{attribute 'pack_mode' := '2'}
TYPE ST_CAM_CTRL :
STRUCT
  eCtrl               : E_AXIS_CTRL;    // commanded axis function
  eProgress           : E_PROGRESS;     // progress command for synced functions
END_STRUCT
END_TYPE

(* stored: Version 1.1.0.1, ProductVersion 3.1.4024.12
   DUT ST_CAM_CTRL: Id {2b4dad11-6d18-0e6f-2be1-3edcadce9751} *)
